{attribute addProperty BoxType "EK1122-0000-0018"}
{attribute addProperty Id "Beckhoff_EPP2xxxsub_EK1100EK1100_179A0949162A_0001_EPP2008_0001_0016EPP2008_A854BE6D8110.125A_0002_EPP2008_0001_0017EPP2008_A854BE6D8110.125A_0003_EPP2008_0001_0018EPP2008_A854BE6D8110.125A_0004_EPP2008_0002_0016EPP2008_A854BE6D8110.125A_0005_EPP2008_0002_0017EPP2008_A854BE6D8110.125A_0006_EPP2008_0002_0018EPP2008_A854BE6D8110.125A_0007_EPP2008_0022_0016EPP2008_A854BE6D8110.125A_0008_EPP2028_0001_0016EPP2028_A854BE6D8110.125A_0009_EPP2028_0001_0017EPP2028_A854BE6D8110.125A_0010_EPP2028_0002_0016EPP2028_A854BE6D8110.125A_0011_EPP2028_0002_0017EPP2028_A854BE6D8110.125A_0012_EPP2038_0001_0016EPP2038_9444C9D314618.25A_0013_EPP2038_0002_0016EPP2038_9444C9D314618.25A_0014_EPP2304_0061_0016EPP2304_B8CEE24B506.25A_0015_EPP2304_0061_0017EPP2304_B8CEE24B506.25A_0016_EPP2304_0061_0018EPP2304_B8CEE24B506.25A_0017_EPP2308_0001_0016EPP2308_97B4DD118210.25A_0018_EPP2308_0001_0017EPP2308_97B4DD118210.25A_0019_EPP2308_0001_0018EPP2308_97B4DD118210.25A_0020_EPP2308_0002_0016EPP2308_97B4DD118210.25A_0021_EPP2308_0002_0017EPP2308_97B4DD118210.25A_0022_EPP2308_0002_0018EPP2308_97B4DD118210.25A_0023_EPP2316_0003_0016EPP2316_7CBF98C533842.25A_0024_EPP2316_0003_0017EPP2316_7CBF98C533842.25A_0025_EPP2316_0003_0018EPP2316_BCC80C6433842.25A_0026_EPP2316_0008_0016EPP2316_7CBF98C533842.25A_0027_EPP2316_0008_0017EPP2316_7CBF98C533842.25A_0028_EPP2316_0008_0018EPP2316_BCC80C6433842.25A_0029_EPP2318_0001_0016EPP2318_97B4DD118210.25A_0030_EPP2318_0001_0017EPP2318_97B4DD118210.25A_0031_EPP2318_0001_0018EPP2318_97B4DD118210.25A_0032_EPP2318_0002_0016EPP2318_97B4DD118210.25A_0033_EPP2318_0002_0017EPP2318_97B4DD118210.25A_0034_EPP2318_0002_0018EPP2318_97B4DD118210.25A_0035_EPP2328_0001_0016EPP2328_97B4DD118210.25A_0036_EPP2328_0001_0017EPP2328_97B4DD118210.25A_0037_EPP2328_0001_0018EPP2328_97B4DD118210.25A_0038_EPP2328_0002_0016EPP2328_97B4DD118210.25A_0039_EPP2328_0002_0017EPP2328_97B4DD118210.25A_0040_EPP2328_0002_0018EPP2328_97B4DD118210.25A_0041_EPP2334_0061_0016EPP2334_97B4DD118210.25A_0042_EPP2334_0061_0017EPP2334_97B4DD118210.25A_0043_EPP2334_0061_0018EPP2334_97B4DD118210.25A_0044_EPP2334_0061_0019EPP2334_97B4DD118210.25A_0045_EPP2338_0001_0016EPP2338_538B459D14618.25A_0046_EPP2338_0001_0017EPP2338_538B459D14618.25A_0047_EPP2338_0001_0018EPP2338_538B459D14618.25A_0048_EPP2338_0002_0016EPP2338_538B459D14618.25A_0049_EPP2338_0002_0017EPP2338_538B459D14618.25A_0050_EPP2338_0002_0018EPP2338_538B459D14618.25A_0051_EPP2338_1001_0017EPP2338_538B459D14618.25A_0052_EPP2338_1001_0018EPP2338_538B459D14618.25A_0053_EPP2338_1001_0019EPP2338_538B459D14618.25A_0054_EPP2338_1002_0017EPP2338_538B459D14618.25A_0055_EPP2338_1002_0018EPP2338_538B459D14618.25A_0056_EPP2338_1002_0019EPP2338_538B459D14618.25A_0057_EPP2339_0003_0016EPP2339_41D05C2438648.25A_0058_EPP2339_0021_0016EPP2339_D38077EA27434.25A_0059_EPP2339_0021_0017EPP2339_9219B49827434.25A_0060_EPP2339_0021_0018EPP2339_9219B49827434.25A_0061_EPP2339_0022_0016EPP2339_D38077EA27434.25A_0062_EPP2339_0022_0017EPP2339_9219B49827434.25A_0063_EPP2339_0022_0018EPP2339_9219B49827434.25A_0064_EPP2349_0021_0016EPP2349_D38077EA27434.25A_0065_EPP2349_0021_0017EPP2349_9219B49827434.25A_0066_EPP2349_0021_0018EPP2349_9219B49827434.25A_0067_EPP2349_0022_0016EPP2349_D38077EA27434.25A_0068_EPP2349_0022_0017EPP2349_9219B49827434.25A_0069_EPP2349_0022_0018EPP2349_9219B49827434.25A_0070_EPP2624_0002_0016EPP2624_4E3C7537496.125A_0071_EPP2809_0021_0016EPP2809_859F43D214518.125A_0072_EPP2809_0022_0016EPP2809_859F43D214518.125A_0073_EPP2816_0004_0016EPP2816_E74B64DB39449.25A_0074_EPP2816_0004_0017EPP2816_E74B64DB39449.25A_0075_EPP2816_0008_0016EPP2816_907EDA0F39449.25A_0076_EPP2816_0008_0017EPP2816_907EDA0F39449.25A_0077_EPP2816_0008_0018EPP2816_56AF2AEC39449.25A_0078_EPP2816_0010_0016EPP2816_907EDA0F39449.25A_0079_EPP2816_0010_0017EPP2816_907EDA0F39449.25A_0080_EPP2816_0010_0018EPP2816_56AF2AEC39449.25A_0081_EPP2817_0008_0016EPP2817_AE3316D954668.25A_0082_EPP2817_0008_0017EPP2817_AE3316D954668.25A_0083_EPP2817_0008_0018EPP2817_AE3316D954668.25"}
{attribute addProperty CRC "212629522"}
{attribute addProperty SizeInBites "15736"}
{attribute addProperty SizeInBytes "1967"}
TYPE Beckhoff_EPP2xxxEK1122_0CAC7812 EXTENDS EK1122_179A0949 :
STRUCT
	{attribute addProperty Name "Beckhoff_EPP2xxxsub_EK1100"}
	Beckhoff_EPP2xxxsub_EK1100 : EK1100_179A0949;
	{attribute addProperty Name "A_0001_EPP2008_0001_0016"}
	A_0001_EPP2008_0001_0016 : EPP2008_A854BE6D;
	{attribute addProperty Name "A_0002_EPP2008_0001_0017"}
	A_0002_EPP2008_0001_0017 : EPP2008_A854BE6D;
	{attribute addProperty Name "A_0003_EPP2008_0001_0018"}
	A_0003_EPP2008_0001_0018 : EPP2008_A854BE6D;
	{attribute addProperty Name "A_0004_EPP2008_0002_0016"}
	A_0004_EPP2008_0002_0016 : EPP2008_A854BE6D;
	{attribute addProperty Name "A_0005_EPP2008_0002_0017"}
	A_0005_EPP2008_0002_0017 : EPP2008_A854BE6D;
	{attribute addProperty Name "A_0006_EPP2008_0002_0018"}
	A_0006_EPP2008_0002_0018 : EPP2008_A854BE6D;
	{attribute addProperty Name "A_0007_EPP2008_0022_0016"}
	A_0007_EPP2008_0022_0016 : EPP2008_A854BE6D;
	{attribute addProperty Name "A_0008_EPP2028_0001_0016"}
	A_0008_EPP2028_0001_0016 : EPP2028_A854BE6D;
	{attribute addProperty Name "A_0009_EPP2028_0001_0017"}
	A_0009_EPP2028_0001_0017 : EPP2028_A854BE6D;
	{attribute addProperty Name "A_0010_EPP2028_0002_0016"}
	A_0010_EPP2028_0002_0016 : EPP2028_A854BE6D;
	{attribute addProperty Name "A_0011_EPP2028_0002_0017"}
	A_0011_EPP2028_0002_0017 : EPP2028_A854BE6D;
	{attribute addProperty Name "A_0012_EPP2038_0001_0016"}
	A_0012_EPP2038_0001_0016 : EPP2038_9444C9D3;
	{attribute addProperty Name "A_0013_EPP2038_0002_0016"}
	A_0013_EPP2038_0002_0016 : EPP2038_9444C9D3;
	{attribute addProperty Name "A_0014_EPP2304_0061_0016"}
	A_0014_EPP2304_0061_0016 : EPP2304_B8CEE24B;
	{attribute addProperty Name "A_0015_EPP2304_0061_0017"}
	A_0015_EPP2304_0061_0017 : EPP2304_B8CEE24B;
	{attribute addProperty Name "A_0016_EPP2304_0061_0018"}
	A_0016_EPP2304_0061_0018 : EPP2304_B8CEE24B;
	{attribute addProperty Name "A_0017_EPP2308_0001_0016"}
	A_0017_EPP2308_0001_0016 : EPP2308_97B4DD11;
	{attribute addProperty Name "A_0018_EPP2308_0001_0017"}
	A_0018_EPP2308_0001_0017 : EPP2308_97B4DD11;
	{attribute addProperty Name "A_0019_EPP2308_0001_0018"}
	A_0019_EPP2308_0001_0018 : EPP2308_97B4DD11;
	{attribute addProperty Name "A_0020_EPP2308_0002_0016"}
	A_0020_EPP2308_0002_0016 : EPP2308_97B4DD11;
	{attribute addProperty Name "A_0021_EPP2308_0002_0017"}
	A_0021_EPP2308_0002_0017 : EPP2308_97B4DD11;
	{attribute addProperty Name "A_0022_EPP2308_0002_0018"}
	A_0022_EPP2308_0002_0018 : EPP2308_97B4DD11;
	{attribute addProperty Name "A_0023_EPP2316_0003_0016"}
	A_0023_EPP2316_0003_0016 : EPP2316_7CBF98C5;
	{attribute addProperty Name "A_0024_EPP2316_0003_0017"}
	A_0024_EPP2316_0003_0017 : EPP2316_7CBF98C5;
	{attribute addProperty Name "A_0025_EPP2316_0003_0018"}
	A_0025_EPP2316_0003_0018 : EPP2316_BCC80C64;
	{attribute addProperty Name "A_0026_EPP2316_0008_0016"}
	A_0026_EPP2316_0008_0016 : EPP2316_7CBF98C5;
	{attribute addProperty Name "A_0027_EPP2316_0008_0017"}
	A_0027_EPP2316_0008_0017 : EPP2316_7CBF98C5;
	{attribute addProperty Name "A_0028_EPP2316_0008_0018"}
	A_0028_EPP2316_0008_0018 : EPP2316_BCC80C64;
	{attribute addProperty Name "A_0029_EPP2318_0001_0016"}
	A_0029_EPP2318_0001_0016 : EPP2318_97B4DD11;
	{attribute addProperty Name "A_0030_EPP2318_0001_0017"}
	A_0030_EPP2318_0001_0017 : EPP2318_97B4DD11;
	{attribute addProperty Name "A_0031_EPP2318_0001_0018"}
	A_0031_EPP2318_0001_0018 : EPP2318_97B4DD11;
	{attribute addProperty Name "A_0032_EPP2318_0002_0016"}
	A_0032_EPP2318_0002_0016 : EPP2318_97B4DD11;
	{attribute addProperty Name "A_0033_EPP2318_0002_0017"}
	A_0033_EPP2318_0002_0017 : EPP2318_97B4DD11;
	{attribute addProperty Name "A_0034_EPP2318_0002_0018"}
	A_0034_EPP2318_0002_0018 : EPP2318_97B4DD11;
	{attribute addProperty Name "A_0035_EPP2328_0001_0016"}
	A_0035_EPP2328_0001_0016 : EPP2328_97B4DD11;
	{attribute addProperty Name "A_0036_EPP2328_0001_0017"}
	A_0036_EPP2328_0001_0017 : EPP2328_97B4DD11;
	{attribute addProperty Name "A_0037_EPP2328_0001_0018"}
	A_0037_EPP2328_0001_0018 : EPP2328_97B4DD11;
	{attribute addProperty Name "A_0038_EPP2328_0002_0016"}
	A_0038_EPP2328_0002_0016 : EPP2328_97B4DD11;
	{attribute addProperty Name "A_0039_EPP2328_0002_0017"}
	A_0039_EPP2328_0002_0017 : EPP2328_97B4DD11;
	{attribute addProperty Name "A_0040_EPP2328_0002_0018"}
	A_0040_EPP2328_0002_0018 : EPP2328_97B4DD11;
	{attribute addProperty Name "A_0041_EPP2334_0061_0016"}
	A_0041_EPP2334_0061_0016 : EPP2334_97B4DD11;
	{attribute addProperty Name "A_0042_EPP2334_0061_0017"}
	A_0042_EPP2334_0061_0017 : EPP2334_97B4DD11;
	{attribute addProperty Name "A_0043_EPP2334_0061_0018"}
	A_0043_EPP2334_0061_0018 : EPP2334_97B4DD11;
	{attribute addProperty Name "A_0044_EPP2334_0061_0019"}
	A_0044_EPP2334_0061_0019 : EPP2334_97B4DD11;
	{attribute addProperty Name "A_0045_EPP2338_0001_0016"}
	A_0045_EPP2338_0001_0016 : EPP2338_538B459D;
	{attribute addProperty Name "A_0046_EPP2338_0001_0017"}
	A_0046_EPP2338_0001_0017 : EPP2338_538B459D;
	{attribute addProperty Name "A_0047_EPP2338_0001_0018"}
	A_0047_EPP2338_0001_0018 : EPP2338_538B459D;
	{attribute addProperty Name "A_0048_EPP2338_0002_0016"}
	A_0048_EPP2338_0002_0016 : EPP2338_538B459D;
	{attribute addProperty Name "A_0049_EPP2338_0002_0017"}
	A_0049_EPP2338_0002_0017 : EPP2338_538B459D;
	{attribute addProperty Name "A_0050_EPP2338_0002_0018"}
	A_0050_EPP2338_0002_0018 : EPP2338_538B459D;
	{attribute addProperty Name "A_0051_EPP2338_1001_0017"}
	A_0051_EPP2338_1001_0017 : EPP2338_538B459D;
	{attribute addProperty Name "A_0052_EPP2338_1001_0018"}
	A_0052_EPP2338_1001_0018 : EPP2338_538B459D;
	{attribute addProperty Name "A_0053_EPP2338_1001_0019"}
	A_0053_EPP2338_1001_0019 : EPP2338_538B459D;
	{attribute addProperty Name "A_0054_EPP2338_1002_0017"}
	A_0054_EPP2338_1002_0017 : EPP2338_538B459D;
	{attribute addProperty Name "A_0055_EPP2338_1002_0018"}
	A_0055_EPP2338_1002_0018 : EPP2338_538B459D;
	{attribute addProperty Name "A_0056_EPP2338_1002_0019"}
	A_0056_EPP2338_1002_0019 : EPP2338_538B459D;
	{attribute addProperty Name "A_0057_EPP2339_0003_0016"}
	A_0057_EPP2339_0003_0016 : EPP2339_41D05C24;
	{attribute addProperty Name "A_0058_EPP2339_0021_0016"}
	A_0058_EPP2339_0021_0016 : EPP2339_D38077EA;
	{attribute addProperty Name "A_0059_EPP2339_0021_0017"}
	A_0059_EPP2339_0021_0017 : EPP2339_9219B498;
	{attribute addProperty Name "A_0060_EPP2339_0021_0018"}
	A_0060_EPP2339_0021_0018 : EPP2339_9219B498;
	{attribute addProperty Name "A_0061_EPP2339_0022_0016"}
	A_0061_EPP2339_0022_0016 : EPP2339_D38077EA;
	{attribute addProperty Name "A_0062_EPP2339_0022_0017"}
	A_0062_EPP2339_0022_0017 : EPP2339_9219B498;
	{attribute addProperty Name "A_0063_EPP2339_0022_0018"}
	A_0063_EPP2339_0022_0018 : EPP2339_9219B498;
	{attribute addProperty Name "A_0064_EPP2349_0021_0016"}
	A_0064_EPP2349_0021_0016 : EPP2349_D38077EA;
	{attribute addProperty Name "A_0065_EPP2349_0021_0017"}
	A_0065_EPP2349_0021_0017 : EPP2349_9219B498;
	{attribute addProperty Name "A_0066_EPP2349_0021_0018"}
	A_0066_EPP2349_0021_0018 : EPP2349_9219B498;
	{attribute addProperty Name "A_0067_EPP2349_0022_0016"}
	A_0067_EPP2349_0022_0016 : EPP2349_D38077EA;
	{attribute addProperty Name "A_0068_EPP2349_0022_0017"}
	A_0068_EPP2349_0022_0017 : EPP2349_9219B498;
	{attribute addProperty Name "A_0069_EPP2349_0022_0018"}
	A_0069_EPP2349_0022_0018 : EPP2349_9219B498;
	{attribute addProperty Name "A_0070_EPP2624_0002_0016"}
	A_0070_EPP2624_0002_0016 : EPP2624_4E3C7537;
	{attribute addProperty Name "A_0071_EPP2809_0021_0016"}
	A_0071_EPP2809_0021_0016 : EPP2809_859F43D2;
	{attribute addProperty Name "A_0072_EPP2809_0022_0016"}
	A_0072_EPP2809_0022_0016 : EPP2809_859F43D2;
	{attribute addProperty Name "A_0073_EPP2816_0004_0016"}
	A_0073_EPP2816_0004_0016 : EPP2816_E74B64DB;
	{attribute addProperty Name "A_0074_EPP2816_0004_0017"}
	A_0074_EPP2816_0004_0017 : EPP2816_E74B64DB;
	{attribute addProperty Name "A_0075_EPP2816_0008_0016"}
	A_0075_EPP2816_0008_0016 : EPP2816_907EDA0F;
	{attribute addProperty Name "A_0076_EPP2816_0008_0017"}
	A_0076_EPP2816_0008_0017 : EPP2816_907EDA0F;
	{attribute addProperty Name "A_0077_EPP2816_0008_0018"}
	A_0077_EPP2816_0008_0018 : EPP2816_56AF2AEC;
	{attribute addProperty Name "A_0078_EPP2816_0010_0016"}
	A_0078_EPP2816_0010_0016 : EPP2816_907EDA0F;
	{attribute addProperty Name "A_0079_EPP2816_0010_0017"}
	A_0079_EPP2816_0010_0017 : EPP2816_907EDA0F;
	{attribute addProperty Name "A_0080_EPP2816_0010_0018"}
	A_0080_EPP2816_0010_0018 : EPP2816_56AF2AEC;
	{attribute addProperty Name "A_0081_EPP2817_0008_0016"}
	A_0081_EPP2817_0008_0016 : EPP2817_AE3316D9;
	{attribute addProperty Name "A_0082_EPP2817_0008_0017"}
	A_0082_EPP2817_0008_0017 : EPP2817_AE3316D9;
	{attribute addProperty Name "A_0083_EPP2817_0008_0018"}
	A_0083_EPP2817_0008_0018 : EPP2817_AE3316D9;
END_STRUCT
END_TYPE

(* stored: Version 1.2.0.0, ProductVersion 3.1.4024.9
   DUT Beckhoff_EPP2xxxEK1122_0CAC7812: Id {804bf46b-a399-4ba7-8458-6dc9e529344e} *)
